TYPE TYP_FAULHABER_SC_HW_IN :
STRUCT
	Fault AT %I*: BOOL;
END_STRUCT
END_TYPE

(* stored: Version 1.1.0.1, ProductVersion 3.1.4024.12
   DUT TYP_FAULHABER_SC_HW_IN: Id {e520052d-5600-42e4-a29e-5e2ca02ef8d9} *)
